// TwinCAT 3 PLC project AdsLogEventExample
// ProgramVersion: 3.1.4023.0
// libraries:
//   Tc2_Standard, * (Beckhoff Automation GmbH)
//   Tc2_System, * (Beckhoff Automation GmbH)
//   Tc3_Module, * (Beckhoff Automation GmbH)
// project tree:
//   DUTs/ ST_EventData.TcDUT
//   POUs/ MAIN.TcPOU
//   / Standard.TcTTO
// real-time tasks:
//   TASK PlcTask: cycle T#10ms, priority 20, ADS port 350
//   TASK VISU_TASK: cycle T#200000us, priority 30, ADS port 351
// motion (NC):
//   TASK NC-Task 1 SAF: cycle T#2ms, priority 4, ADS port 501
//   TASK NC-Task 1 SVB: cycle T#10ms, priority 8, ADS port 511
//   AXIS Axis 1 (id 1)
//     OtherSettings: AllowMotionCmdToSlave=true
//     encoder EncType=1
//     drive DrvType=5
//       Analog: TorqueSetpointScale=10, ScaleFactorActTorque=0.1
//       TimeComp: TaskDelayCycles=1
//     controller CtrType=1
//       CtrPara: PriorControlFactor=1
//         Observer: BandWidth=20
// variable links:
//   Tc3EventLoggerUsage/Tc3EventLoggerUsage Instance <-> NC-Task 1 SAF/Axes/Axis 1
//     PlcTask Inputs/MAIN.Axis.NcToPlc <-> Outputs/ToPlc
//     PlcTask Outputs/MAIN.Axis.PlcToNc <-> Inputs/FromPlc

CONFIGURATION AdsLogEventExample
    RESOURCE PLC ON TwinCAT3
        TASK Standard(INTERVAL := T#10ms, PRIORITY := 20);
        PROGRAM MAIN WITH Standard : MAIN;
    END_RESOURCE
END_CONFIGURATION

// ---- DUTs/ST_EventData.TcDUT
TYPE ST_EventData :
STRUCT
	rVal 	: LREAL;
	iVal	: UDINT;
END_STRUCT
END_TYPE

// ---- POUs/MAIN.TcPOU
PROGRAM MAIN
VAR
	CfgEvent				: TcEvent;
	fbEvent					: ADSLOGEVENT;

	eventData				: ST_EventData;
	TcEventDataFormatString : STRING	:= '%f%d';
END_VAR

CfgEvent.Class := TCEVENTCLASS_ALARM;
CfgEvent.Prio := 2;
CfgEvent.Id := 2;
CfgEvent.SourceId := 102;
CfgEvent.bQuitRequired := CfgEvent.bQuitRequired;
CfgEvent.DataFormatStrAddress := ADR(TcEventDataFormatString);
CfgEvent.Flags := TCEVENTFLAG_LOG OR TCEVENTFLAG_SRCID OR TCEVENTFLAG_AUTOFMTALL;
CfgEvent.StreamType := TCEVENTSTREAM_SIMPLE;
CfgEvent.ProgId :='TcEventFormatter.TcXMLFormatter' ;

eventData.rVal 	:= 2.65;
eventData.iVal	:= 3;


		
fbEvent(
	NETID:= '', 
	PORT:= 110, 
	Event:= fbEvent.Event, 
	EventQuit:= fbEvent.EventQuit, 
	EventConfigData:= CfgEvent, 
	EventDataAddress:= ADR(eventData), 
	EventDataLength:=  SIZEOF(eventData),
	FbCleanup:= , 
	TMOUT:= T#3S, 
	EventState=> , 
	Err=> , 
	ErrId=> , 
	Quit=> );

END_PROGRAM
